Universal Robots PolyScope program: ros_20220917.urp

Program ros_20220917 (installation=default directory=/ursim/programs createdIn=5.12.2.1101534 lastSavedIn=5.12.2.1101534 robotSerialNumber=20195399999)
Calibrated DH parameters: a=[0, -0.24355, -0.2132, 0, 0, 0]; d=[0.15185, 0, 0, 0.13105, 0.08535, 0.0921]; alpha=[1.570796, 0, 0, 1.570796, -1.570796, 0]; deltaTheta=[0, 0, 0, 0, 0, 0]
Robot Program (runOnlyOnce=false)
  Placeholder
